FUNCTION_BLOCK FB_RunningState IMPLEMENTS I_State
VAR_INPUT
END_VAR
VAR_OUTPUT
END_VAR
VAR
	pMachine : POINTER TO FB_StateMachine;	
END_VAR

METHOD ActionSwitchOff : BOOL
VAR_INPUT
	message		:	STRING;
END_VAR
pMachine^.timerTON(IN := TRUE, PT := GVL.configValues.minIdleSec);
ADSLOGSTR(ADSLOG_MSGTYPE_HINT, message, pMachine^.CoolDownState.Name);
pMachine^.pd.actor.operatingStateCompressor := FALSE;
pMachine^.SetState(pMachine^.CoolDownState);
END_METHOD

PROPERTY Description : STRING
GET
Description := 'Heat pump is running';
END_GET
END_PROPERTY

METHOD ErrorDetected : BOOL
VAR_INPUT
	errorEvents		: ST_ErrorEvents;
END_VAR
VAR
	message				: STRING(255);
END_VAR
message := toErrorText(errorEvents);
ADSLOGSTR(ADSLOG_MSGTYPE_HINT, 'Error detected', message);
pMachine^.SetState(pMachine^.ErrorState);
END_METHOD

//FB_Init ist immer implizit verfügbar und wird primär für die Initialisierung verwendet.
//Der Rückgabewert wird nicht ausgewertet. Für gezielte Einflussnahme können Sie
//die Methoden explizit deklarieren und darin mit dem Standard-Initialisierungscode 
//zusätzlichen Code bereitstellen. Sie können den Rückgabewert auswerten.
METHOD FB_Init: BOOL
VAR_INPUT    
	bInitRetains: BOOL; // TRUE: Die Retain-Variablen werden initialisiert (Reset warm / Reset kalt)    
	bInCopyCode: BOOL;  // TRUE: Die Instanz wird danach in den Kopiercode kopiert (Online-Change)
	pMachine : POINTER TO FB_StateMachine;
END_VAR
THIS^.pMachine := pMachine;
END_METHOD

METHOD HeatIsRequested : BOOL
END_METHOD

METHOD LimitValuesAreExceeded : BOOL
END_METHOD

PROPERTY Name : STRING
GET
Name := 'Running';
END_GET
END_PROPERTY

PROPERTY State : E_State
GET
State := E_State.RUNNING;
END_GET
END_PROPERTY

METHOD TargetTemeperatureReached : BOOL
ActionSwitchOff('Zieltemperatur erreicht. -> %s');
END_METHOD

METHOD UserPressedConfirmationButton : BOOL
END_METHOD

METHOD UserPressedSwitchOffButton : BOOL
ActionSwitchOff('Off Button pressed -> %s');
END_METHOD

METHOD UserPressedSwitchOnButton : BOOL
END_METHOD

METHOD WaterHasCooledDown : BOOL
END_METHOD

END_FUNCTION_BLOCK

(* stored: Version 1.1.0.1
   POU FB_RunningState: Id {db7d51fb-2638-4812-b81a-d21aedf1ed00}, SpecialFunc None
   Method ActionSwitchOff: Id {46ba5a55-86e3-4497-8746-3df853385ea5}
   Property Description: Id {fff56124-f3e0-4a4a-810d-d034fa66ff15}
   Get Get: Id {09f84e37-527b-4c45-880e-5502fab1a5a1}
   Method ErrorDetected: Id {2d6db66f-da00-40a1-96dd-ed61a3c7e83c}
   Method FB_init: Id {ccdf553b-48e7-41c3-825a-9b44d85c7b93}
   Method HeatIsRequested: Id {a0b9eadd-22d5-49b2-8876-9665b4185501}
   Method LimitValuesAreExceeded: Id {ad40b40e-36c5-4eb1-933c-96726184bd4b}
   Property Name: Id {4e96be48-1bba-4ddc-ae4e-db1f900e7cdf}
   Get Get: Id {7e39c09e-d876-4302-9bbd-d2a517af0670}
   Property State: Id {75386ad7-2492-4d3c-8098-8f6c395c0bbb}
   Get Get: Id {81495c4a-f76d-4331-90b6-4378394cf226}
   Method TargetTemeperatureReached: Id {5a9d8a2b-41ae-4ad4-8cdf-a0d67cc0af04}
   Method UserPressedConfirmationButton: Id {34138e8e-29b3-43c6-83b9-21f3a75e6954}
   Method UserPressedSwitchOffButton: Id {f7bc4756-a2f3-4317-96b9-0b7e1640f0e8}
   Method UserPressedSwitchOnButton: Id {92d0b6bf-2822-477d-9e93-031fae1f4a37}
   Method WaterHasCooledDown: Id {58ca67bc-c547-44a6-8e50-bdee1b3ac7d1} *)
